FUNCTION_BLOCK EdgeDetector
VAR_INPUT
	inputValue : BOOL ;
END_VAR

VAR_OUTPUT
	riesingEdge :BOOL;
	fallingEdge :BOOL;
END_VAR
VAR
	safeStatus:BOOL;
END_VAR



IF safeStatus = FALSE AND inputValue = TRUE THEN
riesingEdge:= TRUE;
fallingEdge:= FALSE;
ELSIF safeStatus = TRUE AND inputValue = FALSE THEN
fallingEdge:= TRUE;
riesingEdge:= FALSE;
END_IF
safeStatus := inputValue;

END_FUNCTION_BLOCK

(* stored: Version 1.1.0.1, ProductVersion 3.1.4022.12
   POU EdgeDetector: Id {20a7cb78-1e55-4a66-9642-d8d122f25561}, SpecialFunc None *)
